TYPE AX5000_P_0209 :
STRUCT
	Internal_brak_resistor_actual_continouse_power:UINT;
END_STRUCT
END_TYPE

(* stored: Version 1.1.0.1, ProductVersion 3.1.4024.3
   DUT AX5000_P_0209: Id {4628588f-ba6b-4384-bab9-f6d54887a718} *)
